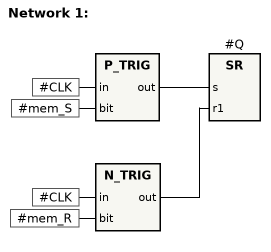
   #_w1 := #CLK AND NOT #mem_S;   // rising edge
   #mem_S := #CLK;
   #_w2 := NOT #CLK AND #mem_R;   // falling edge
   #mem_R := #CLK;
   IF #_w1 THEN
       #Q := TRUE;   // SR flip-flop
   END_IF;
   IF #_w2 THEN #Q := FALSE; END_IF;
END_REGION
END_FUNCTION_BLOCK

FUNCTION_BLOCK "TON_seconds"   // FB8, FBD
{ S7_Optimized_Access := 'TRUE' }
VERSION : 0.1
// stored: AutoNumber true, IsIECCheckEnabled false, IsRetainMemResEnabled false, MemoryReserve 100, SetENOAutomatically false, UDAEnableTagReadback false
   VAR_INPUT
      IN : Bool;
      PT_s : DInt;
   END_VAR
   VAR_OUTPUT
      Q : Bool;
   END_VAR
   VAR
      ton { S7_SetPoint := 'True'} : TON_TIME;
   END_VAR
   VAR_TEMP
      PT : Time;
   END_VAR
BEGIN

REGION Network 1
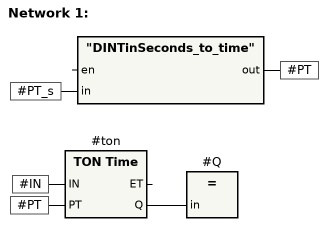
   "DINTinSeconds_to_time"(in := #PT_s, out => #PT);
   #ton(IN := #IN, PT := #PT);   // TON
   #Q := #ton.Q;
END_REGION
END_FUNCTION_BLOCK

FUNCTION_BLOCK "cooling"   // FB17, LAD
{ S7_Optimized_Access := 'TRUE' }
VERSION : 0.1
// stored: AutoNumber true, IsIECCheckEnabled false, IsRetainMemResEnabled false, MemoryReserve 100, SetENOAutomatically false, UDAEnableTagReadback false
   VAR_INPUT
      MagsOn : Bool;
      Work_time_for_CD : Time := T#10m;
   END_VAR
   VAR_OUTPUT
      Vents : Bool;
   END_VAR
   VAR
      IEC_Timer_0_Instance { S7_SetPoint := 'True'} : TON_TIME;
      wasActive : Bool;
   END_VAR
BEGIN

REGION Network 1
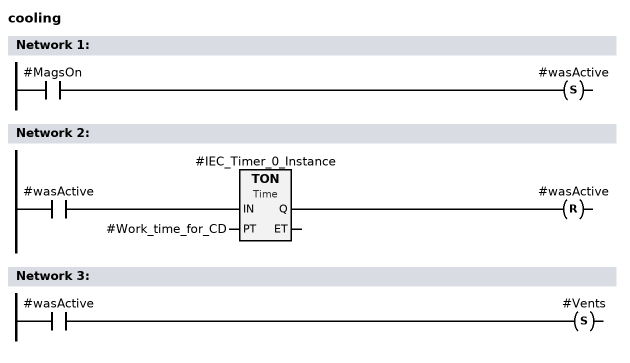
   RUNG wire#powerrail
      Contact( #MagsOn )
      S_Coil( #wasActive )
   END_RUNG
   // the same network as SCL:
   IF #MagsOn THEN #wasActive := TRUE; END_IF;
END_REGION

REGION Network 2
   RUNG wire#powerrail
      Contact( #wasActive )
      { S7_Templates := "time_type := Time" } #IEC_Timer_0_Instance.TON(pt := #Work_time_for_CD, et =>)
      R_Coil( #wasActive )
   END_RUNG
   // the same network as SCL:
   #IEC_Timer_0_Instance(IN := #wasActive, PT := #Work_time_for_CD);   // TON
   IF #IEC_Timer_0_Instance.Q THEN #wasActive := FALSE; END_IF;
END_REGION

REGION Network 3
   RUNG wire#powerrail
      Contact( #wasActive )
      S_Coil( #Vents )
   END_RUNG
   // the same network as SCL:
   IF #wasActive THEN #Vents := TRUE; END_IF;
END_REGION
END_FUNCTION_BLOCK

FUNCTION "LT_GT_OK" : Void   // FC16, FBD
{ S7_Optimized_Access := 'TRUE' }
VERSION : 0.1
// stored: AutoNumber true, IsIECCheckEnabled false, SetENOAutomatically false, UDAEnableTagReadback false
   VAR_INPUT
      value : Real;
      min : Real;
      max : Real;
   END_VAR
   VAR_OUTPUT
      OK : Bool;
      LT_MIN : Bool;
      GT_MAX : Bool;
   END_VAR
BEGIN

REGION Network 1
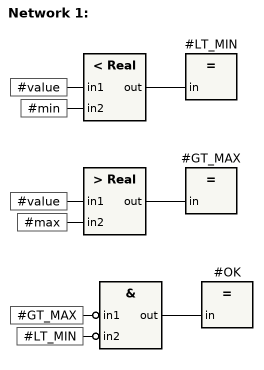
   #LT_MIN := #value < #min;
   #GT_MAX := #value > #max;
   #OK := NOT #GT_MAX AND NOT #LT_MIN;
END_REGION
END_FUNCTION

FUNCTION_BLOCK "execute_semiauto"   // FB46, FBD
{ S7_Optimized_Access := 'TRUE' }
VERSION : 0.1
// stored: AutoNumber true, IsIECCheckEnabled false, IsRetainMemResEnabled false, MemoryReserve 100, SetENOAutomatically false, UDAEnableTagReadback false
   VAR_INPUT
      ALLOWED : Bool;
      xButton : Bool;
      arrived : Bool;
   END_VAR
   VAR_OUTPUT
      y_exec : Bool;
   END_VAR
   VAR
      mem : Bool;
      R_TRIG_Instance { S7_SetPoint := 'True'} : R_TRIG;
      loc : Bool;
   END_VAR
BEGIN

REGION Network 2 (SCL)
   #R_TRIG_Instance(CLK := #xButton);
   IF #ALLOWED THEN
       #y_exec := true;
   (*    IF #R_TRIG_Instance.Q THEN
           IF NOT #arrived THEN
               #y_exec := true;
           ELSE
               #y_exec := false;
           END_IF;
       END_IF; *)
   ELSE
       #y_exec := false;
   END_IF;
END_REGION
END_FUNCTION_BLOCK

FUNCTION_BLOCK "_screen_SetHome"   // FB77, FBD
{ S7_Optimized_Access := 'TRUE' }
VERSION : 0.1
// stored: AutoNumber true, IsIECCheckEnabled false, IsRetainMemResEnabled false, MemoryReserve 100, SetENOAutomatically false, UDAEnableTagReadback false
   VAR
      t_z : "hmi_home_1";
      t_o1 : "hmi_home_1";
      t_o2 : "hmi_home_1";
      t_x : "hmi_home_1";
      t_y : "hmi_home_1";
      z : "hmi_home_1";
      o1 : "hmi_home_1";
      o2 : "hmi_home_1";
      x : "hmi_home_1";
      y : "hmi_home_1";
   END_VAR
BEGIN

REGION Network 1
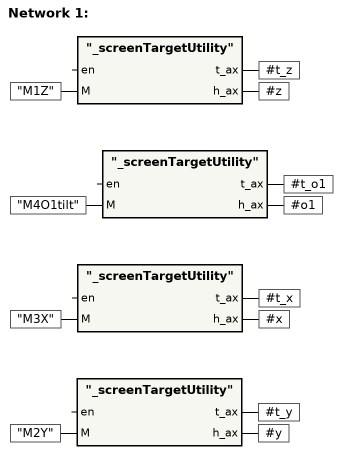
   "_screenTargetUtility"("M" := "M1Z", t_ax => #t_z, h_ax => #z);
   "_screenTargetUtility"("M" := "M4O1tilt", t_ax => #t_o1, h_ax => #o1);
   "_screenTargetUtility"("M" := "M3X", t_ax => #t_x, h_ax => #x);
   "_screenTargetUtility"("M" := "M2Y", t_ax => #t_y, h_ax => #y);
END_REGION

REGION Network 2 (SCL)
   #o2.eF := NOT "M5O2rot".xPredifCal;
   #o2.pos := "M5O2rot".POS;
   #t_o2.pos := "M5O2rot".AMANGRDB.aut_target;
END_REGION
END_FUNCTION_BLOCK

FUNCTION_BLOCK "DelayDirChange"   // FB61, FBD
{ S7_Optimized_Access := 'TRUE' }
VERSION : 0.1
// stored: AutoNumber true, IsIECCheckEnabled false, IsRetainMemResEnabled false, MemoryReserve 100, SetENOAutomatically false, UDAEnableTagReadback false
   VAR_INPUT
      pt : Time := T#2S;
      dirFwd : Bool;
      dirRev : Bool;
   END_VAR
   VAR_OUTPUT
      qFwd : Bool;
      qRev : Bool;
      block : Bool;
   END_VAR
   VAR
      tonfwd { S7_SetPoint := 'True'} : TON_TIME;
      tonrev { S7_SetPoint := 'True'} : TON_TIME;
      block_fwd : Bool;
   END_VAR
   VAR_TEMP
      wait_done : Bool;
      block_rev : Bool;
   END_VAR
BEGIN

REGION Network 2
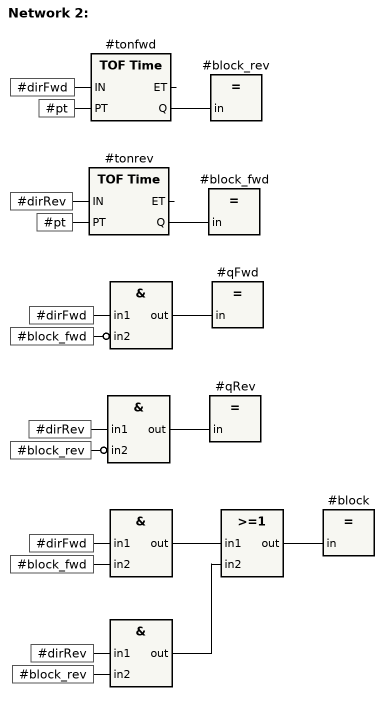
   #tonfwd(IN := #dirFwd, PT := #pt);   // TOF
   #block_rev := #tonfwd.Q;
   #tonrev(IN := #dirRev, PT := #pt);   // TOF
   #block_fwd := #tonrev.Q;
   #qFwd := #dirFwd AND NOT #block_fwd;
   #qRev := #dirRev AND NOT #block_rev;
   #block := (#dirFwd AND #block_fwd) OR (#dirRev AND #block_rev);
END_REGION
END_FUNCTION_BLOCK

FUNCTION_BLOCK "FPDRxMonitorTwoEncodersFB"   // FB63, FBD
{ S7_Optimized_Access := 'TRUE' }
VERSION : 0.1
// stored: AutoNumber true, IsIECCheckEnabled false, IsRetainMemResEnabled false, MemoryReserve 100, SetENOAutomatically false, UDAEnableTagReadback false
   VAR_INPUT
      pos1 { ExternalAccessible := 'False'; ExternalVisible := 'False'; ExternalWritable := 'False'} : Real;
      pos2 { ExternalAccessible := 'False'; ExternalVisible := 'False'; ExternalWritable := 'False'} : Real;
      allowedDelta { ExternalAccessible := 'False'; ExternalVisible := 'False'; ExternalWritable := 'False'} : Real;
      pt : Time;
   END_VAR
   VAR_OUTPUT
      error { ExternalAccessible := 'False'; ExternalVisible := 'False'; ExternalWritable := 'False'} : Bool;
   END_VAR
   VAR
      tonER { S7_SetPoint := 'True'} : TON_TIME;
   END_VAR
   VAR_TEMP
      deltaDangerous : Bool;
   END_VAR
BEGIN

REGION Network 2 (SCL)
   #deltaDangerous := ABS(#pos2 - #pos1)> #allowedDelta;
END_REGION

REGION Network 3
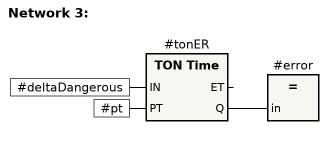
   #tonER(IN := #deltaDangerous, PT := #pt);   // TON
   #error := #tonER.Q;
END_REGION
END_FUNCTION_BLOCK

FUNCTION_BLOCK "Select_remote_or_auto"   // FB24, FBD
{ S7_Optimized_Access := 'TRUE' }
VERSION : 0.1
// stored: AutoNumber true, IsIECCheckEnabled false, IsRetainMemResEnabled false, MemoryReserve 100, SetENOAutomatically false, UDAEnableTagReadback false
BEGIN
END_FUNCTION_BLOCK

FUNCTION_BLOCK "SetA2"   // FB23, FBD
{ S7_Optimized_Access := 'TRUE' }
VERSION : 0.1
// stored: AutoNumber true, IsIECCheckEnabled false, IsRetainMemResEnabled false, MemoryReserve 100, SetENOAutomatically false, UDAEnableTagReadback false
   VAR_INPUT
      xCalibSwMaster : Bool;
      xCalibSwSlave : Bool;
      parMasterCalibPos : Real;
      parSlaveCalibPos : Real;
      btnCopyMasterNow : Bool;
      btnAdjustHorizonPlusStep : Bool;
      btnAdjustHorizonMinusStep : Bool;
      MasterPos : Real;
      SlavePos : Real;
      StepHorAdjust : Real := 10.0;
   END_VAR
   VAR_OUTPUT
      MasterCalibPos : Real;
      MasterCalibNow : Bool;
      SlaveCalibPos : Real;
      SlaveCalibNow : Bool;
   END_VAR
   VAR
      CorrectionFactor : Bool;
      ton { S7_SetPoint := 'True'} : TON_TIME;
      ton1 { S7_SetPoint := 'True'} : TON_TIME;
   END_VAR
BEGIN

REGION Network 1
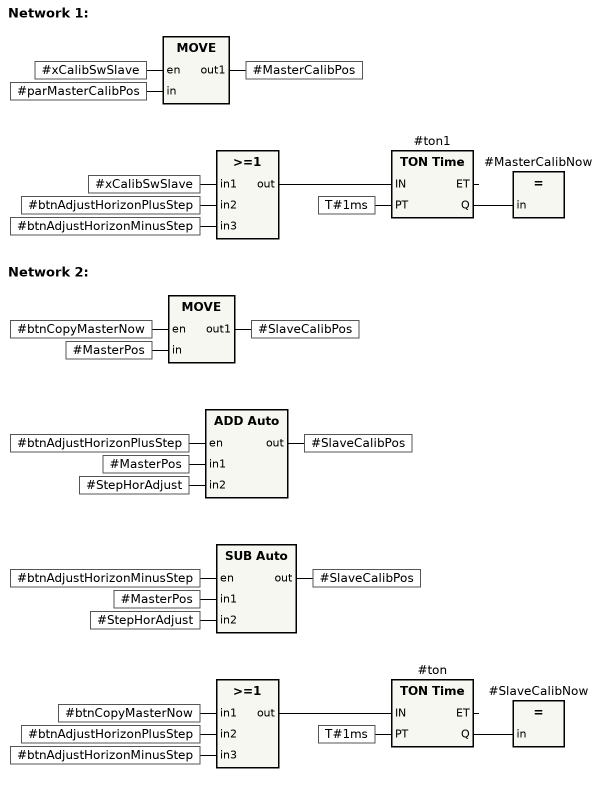
   IF #xCalibSwSlave THEN #MasterCalibPos := #parMasterCalibPos; END_IF;
   #ton1(IN := #xCalibSwSlave OR #btnAdjustHorizonPlusStep OR #btnAdjustHorizonMinusStep, PT := T#1ms);   // TON
   #MasterCalibNow := #ton1.Q;
END_REGION

REGION Network 2
   IF #btnCopyMasterNow THEN #SlaveCalibPos := #MasterPos; END_IF;
   IF #btnAdjustHorizonPlusStep THEN #SlaveCalibPos := #MasterPos + #StepHorAdjust; END_IF;
   IF #btnAdjustHorizonMinusStep THEN #SlaveCalibPos := #MasterPos - #StepHorAdjust; END_IF;
   #ton(IN := #btnCopyMasterNow OR #btnAdjustHorizonPlusStep OR #btnAdjustHorizonMinusStep, PT := T#1ms);   // TON
   #SlaveCalibNow := #ton.Q;
END_REGION
END_FUNCTION_BLOCK

FUNCTION_BLOCK "Slow_inc_quick_drop"   // FB50, FBD
{ S7_Optimized_Access := 'TRUE' }
VERSION : 0.1
// stored: AutoNumber true, IsIECCheckEnabled false, IsRetainMemResEnabled false, MemoryReserve 100, SetENOAutomatically false, UDAEnableTagReadback false
   VAR_INPUT
      ALLOWED : Bool;
      max_v : Real;
      sec_to_max_v : Real;
      req_v : Real;
   END_VAR
   VAR_OUTPUT
      speed : Real;
      er_set { ExternalAccessible := 'False'; ExternalVisible := 'False'; ExternalWritable := 'False'} : Bool;
      wsER : WString;
   END_VAR
   VAR
      accel_v_p_sec : Real;
      accel_per_cycle : Real;
      cycle_time_sec : Real := 0.01;
   END_VAR
BEGIN

REGION Network 2 (SCL)


   #er_set :=  "_MAIN_DB".CLOCK_S_P_SCAN <= 0 OR #sec_to_max_v <=0 ;
   IF #er_set THEN
       #wsER := WSTRING#'ошибка модуля ускорения';
   ELSE
       #wsER := WSTRING#'';
   END_IF;
END_REGION

REGION Network 3 (SCL)
   IF NOT #er_set THEN
       #accel_v_p_sec := #max_v / #sec_to_max_v;
       #accel_per_cycle := #accel_v_p_sec * "_MAIN_DB".CLOCK_S_P_SCAN;
   ELSE
       #accel_per_cycle := 0.0001;
   END_IF;
END_REGION

REGION Network 4 (SCL)
   IF #ALLOWED THEN
       IF NOT #er_set THEN
           IF #req_v > #speed THEN
               #speed := MIN(IN1 := #speed + #accel_per_cycle, IN2 := #req_v);
           ELSIF #req_v < #speed THEN
               #speed := MAX(IN1 := #speed - #accel_per_cycle, IN2 := #req_v);
           END_IF;

       ELSE
           #speed := 0;
       END_IF;
   ELSE
       #speed := 0;
   END_IF;
END_REGION
END_FUNCTION_BLOCK

FUNCTION_BLOCK "auto_digital"   // FB12, FBD
{ S7_Optimized_Access := 'TRUE' }
VERSION : 0.1
// stored: AutoNumber true, IsIECCheckEnabled false, IsRetainMemResEnabled false, MemoryReserve 100, SetENOAutomatically false, UDAEnableTagReadback false
   VAR_INPUT
      ALLOWED : Bool;
      xFwdOK : Bool;
      xRevOK : Bool;
      xFwdFastOK : Bool;
      xRevFastOK : Bool;
   END_VAR
   VAR_OUTPUT
      FWD : Bool;
      REV : Bool;
      QUICK : Bool;
      status_fwd_full : Bool;
      status_mid : Bool;
      status_rev_full : Bool;
   END_VAR
   VAR_IN_OUT
      btn_go_fwd : Bool;
      btn_go_rev : Bool;
   END_VAR
   VAR
      lbs { S7_SetPoint := 'True'} : "last_button_stands";
      mem_fwdok : Bool;
      mem_revok : Bool;
      ton_quick { S7_SetPoint := 'True'} : TON_TIME;
   END_VAR
BEGIN

REGION Network 1
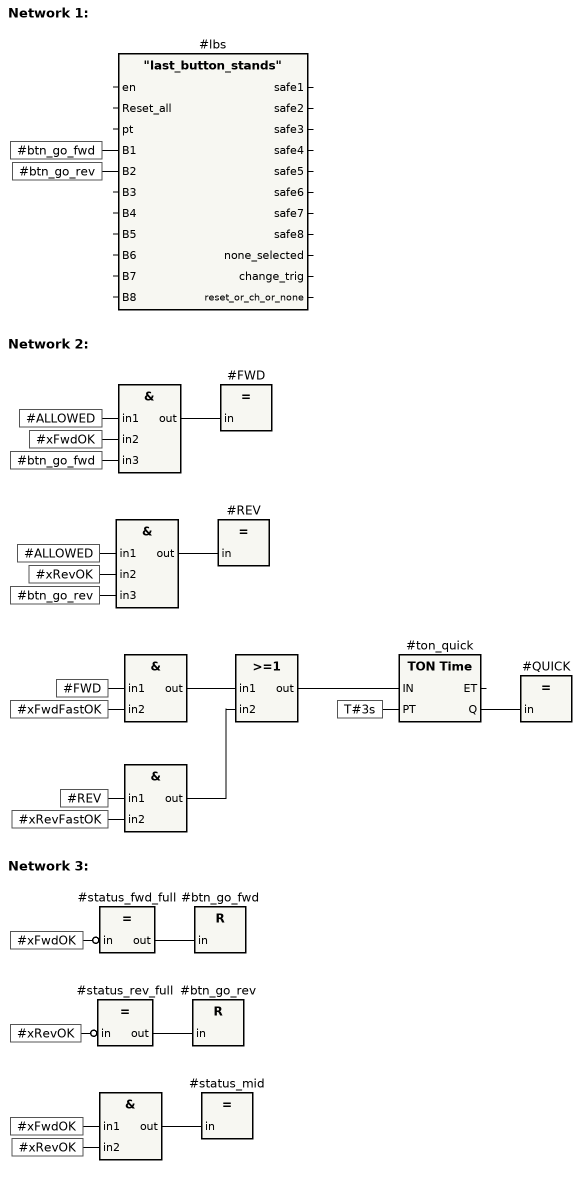
   #lbs(B1 := #btn_go_fwd, B2 := #btn_go_rev);   // "last_button_stands"
END_REGION

REGION Network 2
   #FWD := #ALLOWED AND #xFwdOK AND #btn_go_fwd;
   #REV := #ALLOWED AND #xRevOK AND #btn_go_rev;
   #ton_quick(IN := (#FWD AND #xFwdFastOK) OR (#REV AND #xRevFastOK), PT := T#3s);   // TON
   #QUICK := #ton_quick.Q;
END_REGION

REGION Network 3
   #status_fwd_full := NOT #xFwdOK;
   IF NOT #xFwdOK THEN #btn_go_fwd := FALSE; END_IF;
   #status_rev_full := NOT #xRevOK;
   IF NOT #xRevOK THEN #btn_go_rev := FALSE; END_IF;
   #status_mid := #xFwdOK AND #xRevOK;
END_REGION
END_FUNCTION_BLOCK

FUNCTION "calc_speeds_from_mechanics_1StepperMotor" : Void   // FC33, FBD
{ S7_Optimized_Access := 'TRUE' }
VERSION : 0.1
// stored: AutoNumber true, IsIECCheckEnabled false, SetENOAutomatically false, UDAEnableTagReadback false
   VAR_INPUT
      Vabsmax_deg_per_s : Real;
   END_VAR
   VAR_OUTPUT
      ER_params : Bool;
   END_VAR
   VAR_IN_OUT
      para : "typeMotPara";
   END_VAR
   VAR_TEMP
      counts_per_deg : Real;
      t_acceleration_s : Real;
      "a" : Real;
      v_abs_max : Real;
      t_mx : Real;
      v_min_viable : Real;
      dist_stop : Real;
      dist_auto_done : Real;
      K_min : Real;
      K_min_dist : Real;
      dist_absMax : Real;
   END_VAR
BEGIN

REGION Network 1 (SCL)
   #v_abs_max := #Vabsmax_deg_per_s;
   #t_acceleration_s := #para.t_acc_50Hz_USER;

   #K_min := 0.5 / 50.0;
   #v_min_viable := #v_abs_max * #K_min;

   #t_mx := #t_acceleration_s;
   #ER_params := #t_acceleration_s = 0 OR #v_abs_max = 0 OR #t_mx =0 ;
   IF NOT #ER_params THEN
       #a := #v_abs_max / #t_mx;
       #dist_absMax := #a * #t_mx * #t_mx / 2 + #v_min_viable * #t_mx;
   ELSE
       #a := 0;
        #dist_absMax := 999;
   END_IF;
   #K_min_dist :=0.5/ 50.0 ;//#K_min * 0.8;
   #dist_stop := #dist_absMax * #K_min_dist;
   #dist_auto_done := #dist_stop * 1.2;
END_REGION

REGION Network 2 (SCL)
   //#para.dist_absMax_LOGIC := #dist_fast;
   #para.dist_stop_USER := #dist_stop;
   #para.dist_auto_done_LOGIC := #dist_auto_done;
   //#para.dist_auto_maxCor_LOGIC := 0.1 * #para.dist_absMax_LOGIC;
   #para.v_absoluteMax_LOGIC := #v_abs_max;
   #para.v_crawl_USER := #v_min_viable;
   //#para.v_auto_maxCor_LOGIC := 0.1 * #para.v_absoluteMax_LOGIC;
END_REGION
END_FUNCTION

FUNCTION "calc_speeds_from_mechanics_2SyncedDrivesTUBEZ" : Void   // FC25, FBD
{ S7_Optimized_Access := 'TRUE' }
VERSION : 0.1
// stored: AutoNumber true, IsIECCheckEnabled false, SetENOAutomatically false, UDAEnableTagReadback false
   VAR_INPUT
      mm_per_outputshaft_rev : Real;
      reduction_ration : Real;
      max_revs_at_10V : Real;
      counts_per_encoder_rev : Real;
      encoder_placed_on_motor : Bool;
   END_VAR
   VAR_OUTPUT
      Vabsmax_mm_per_s : Real;
      counts_per_mm : Real;
      ER_params : Bool;
   END_VAR
   VAR_IN_OUT
      para : "typeMotPara";
   END_VAR
   VAR_TEMP
      t_acceleration_s : Real;
      maxV_mm_per_min : Real;
      "a" : Real;
      v_abs_max : Real;
      t_mx : Real;
      dist_fast : Real;
      v_min_viable : Real;
      dist_stop : Real;
      dist_auto_done : Real;
      K_min : Real;
      K_min_dist : Real;
      dist_absMax : Real;
      t_fst : Real;
      v_fast : Real;
   END_VAR
BEGIN

REGION Network 2 (SCL)

   #maxV_mm_per_min := #max_revs_at_10V / #reduction_ration * #mm_per_outputshaft_rev;

   #Vabsmax_mm_per_s := #maxV_mm_per_min / 60;
END_REGION

REGION Network 3 (SCL)
   IF #encoder_placed_on_motor THEN
       #counts_per_mm :=  #counts_per_encoder_rev * #reduction_ration / #mm_per_outputshaft_rev  ;
   ELSE
       #counts_per_mm := #counts_per_encoder_rev /  #mm_per_outputshaft_rev;

   END_IF;
END_REGION

REGION Network 4 (SCL)
   #v_abs_max := #Vabsmax_mm_per_s;
   #t_acceleration_s := #para.t_acc_50Hz_USER;
   #v_fast := #para.v_absoluteMax_LOGIC;

   #K_min := 1.0/50.0;
   #v_min_viable := #v_abs_max * #K_min;

   #t_mx := #t_acceleration_s;
   #ER_params := #t_acceleration_s = 0 OR #v_abs_max = 0 OR #t_mx =0 ;
   IF NOT #ER_params THEN
       #t_fst := #t_acceleration_s * #v_fast / #v_abs_max;
       #a := #v_abs_max / #t_mx;
       #dist_absMax := #a * #t_mx * #t_mx / 2 + #v_min_viable * #t_mx;
       #dist_fast := #a * #t_fst * #t_fst / 2 + #v_min_viable * #t_fst;
   ELSE
       #a := 0;
       #dist_fast := #dist_absMax := 999;
       #t_fst := 0;
   END_IF;
   #K_min_dist := 1.0/ 50.0;//#K_min * 0.8;
   #dist_stop := #dist_absMax * #K_min_dist;
   #dist_auto_done := #dist_stop * 4.0;//1.4;//.0;// 1.2;
END_REGION

REGION Network 5 (SCL)
   #para.dist_absMax_LOGIC := #dist_fast;
   #para.dist_stop_USER := #dist_stop;
   #para.dist_auto_done_LOGIC := #dist_auto_done;
   #para.v_absoluteMax_LOGIC := #v_abs_max;
   #para.v_crawl_USER := #v_min_viable;
END_REGION
END_FUNCTION

FUNCTION_BLOCK "encoder2"   // FB62, FBD
{ S7_Optimized_Access := 'TRUE' }
VERSION : 0.1
// stored: AutoNumber true, IsIECCheckEnabled false, IsRetainMemResEnabled false, MemoryReserve 100, SetENOAutomatically false, UDAEnableTagReadback false
   VAR_INPUT
      xCal : Bool;
      ENC : Real;
      posCal : Real;
   END_VAR
   VAR_OUTPUT
      i_times_cal : Int;
      retain_test : Bool;
      POS : Real;
   END_VAR
   VAR
      xCal_filtered : Bool;
      not_first_scan : Bool;
      offset : Real;
   END_VAR
   VAR RETAIN
      MEM : Real;
   END_VAR
   VAR
      xCal_mem : Bool;
   END_VAR
   VAR RETAIN
      calibrated : Bool;
   END_VAR
   VAR
      ton_block_calib { S7_SetPoint := 'True'} : TON_TIME;
      tonFilter { S7_SetPoint := 'True'} : TON_TIME;
   END_VAR
BEGIN

REGION Network 1
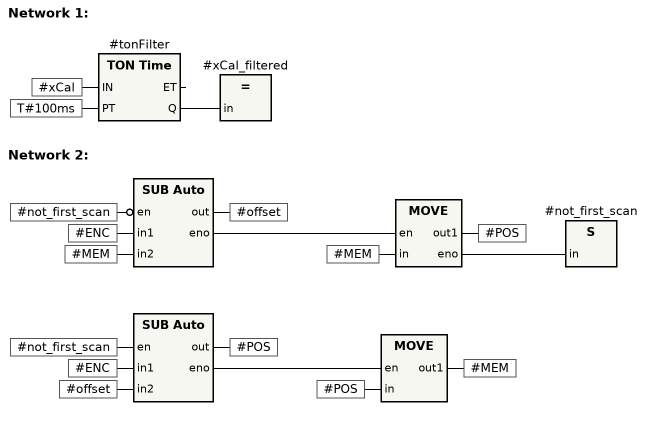
   #tonFilter(IN := #xCal, PT := T#100ms);   // TON
   #xCal_filtered := #tonFilter.Q;
END_REGION

REGION Network 2
   IF NOT #not_first_scan THEN
       #offset := #ENC - #MEM;
       #POS := #MEM;
       #not_first_scan := TRUE;
   END_IF;
   IF #not_first_scan THEN
       #POS := #ENC - #offset;
       #MEM := #POS;
   END_IF;
END_REGION

REGION Network 3 (SCL)
   IF #xCal_filtered AND NOT #xCal_mem THEN
       #offset := #ENC - #posCal;
       #calibrated := true;
       #i_times_cal := #i_times_cal + 1;
   END_IF;
   #xCal_mem := #xCal_filtered;
END_REGION
END_FUNCTION_BLOCK

FUNCTION_BLOCK "encoderMesSpeed"   // FB19, FBD
{ S7_Optimized_Access := 'TRUE' }
VERSION : 0.1
// stored: AutoNumber true, IsIECCheckEnabled false, IsRetainMemResEnabled false, MemoryReserve 100, SetENOAutomatically false, UDAEnableTagReadback false
BEGIN
END_FUNCTION_BLOCK

FUNCTION_BLOCK "encoder_mes_speed"   // FB20, FBD
{ S7_Optimized_Access := 'TRUE' }
VERSION : 0.1
// stored: AutoNumber true, IsIECCheckEnabled false, IsRetainMemResEnabled false, MemoryReserve 100, SetENOAutomatically false, UDAEnableTagReadback false
   VAR_INPUT
      Cycle_Time_s : Real;
      Pos : Real;
   END_VAR
   VAR_OUTPUT
      Speed_mm_p_sec : Real;
   END_VAR
   VAR
      MEM : LReal;
      RET_VAL : LReal;
      Pos_was : Real;
   END_VAR
   VAR_TEMP
      Speed_mm_p_sec_temp : Real;
      delta : Real;
      n : Real;
   END_VAR
BEGIN

REGION Network 1
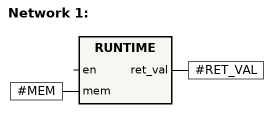
   // no SCL statement known for Runtime: written as a call
   #RET_VAL := Runtime(mem := #MEM);
END_REGION

REGION Network 2 (SCL)
   #delta := #Pos - #Pos_was;
   #Speed_mm_p_sec_temp := #delta / #Cycle_Time_s;
   #n := 10;
   #Speed_mm_p_sec := (#Speed_mm_p_sec * (#n - 1) + #Speed_mm_p_sec_temp)/ #n;

   #Pos_was := #Pos;
END_REGION
END_FUNCTION_BLOCK

FUNCTION_BLOCK "manual_digital"   // FB13, FBD
{ S7_Optimized_Access := 'TRUE' }
VERSION : 0.1
// stored: AutoNumber true, IsIECCheckEnabled false, IsRetainMemResEnabled false, MemoryReserve 100, SetENOAutomatically false, UDAEnableTagReadback false
   VAR_INPUT
      ALLOWED : Bool;
      xFwdOk : Bool;
      xRevOk : Bool;
      xFwdFastOK : Bool;
      xRevFastOK : Bool;
   END_VAR
   VAR_OUTPUT
      FWD : Bool;
      REV : Bool;
      FAST : Bool;
   END_VAR
   VAR_IN_OUT
      btn_FWD : Bool;
      btn_REV : Bool;
   END_VAR
   VAR
      lbs { S7_SetPoint := 'True'} : "last_button_stands";
      ton_quick { S7_SetPoint := 'True'} : TON_TIME;
   END_VAR
BEGIN

REGION Network 1
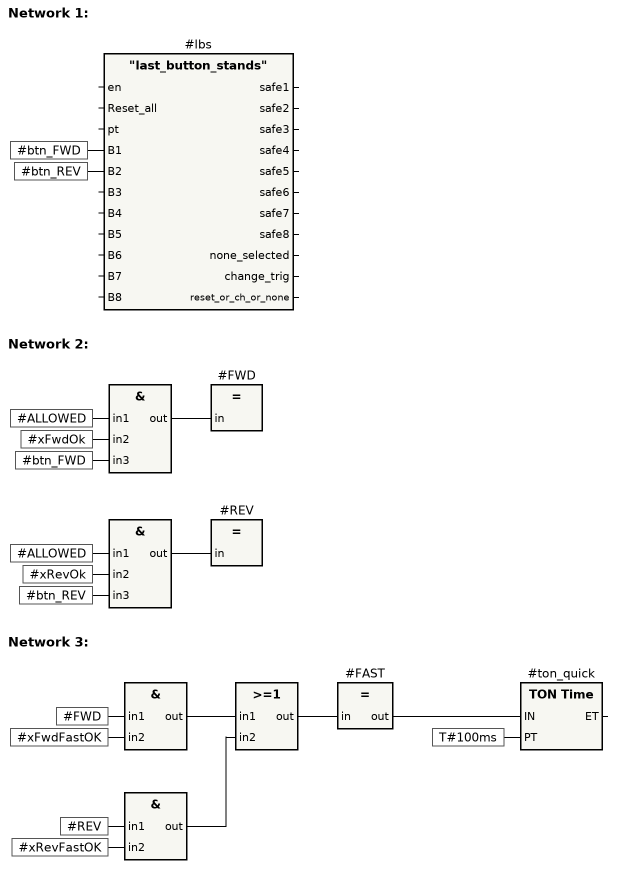
   #lbs(B1 := #btn_FWD, B2 := #btn_REV);   // "last_button_stands"
END_REGION

REGION Network 2
   #FWD := #ALLOWED AND #xFwdOk AND #btn_FWD;
   #REV := #ALLOWED AND #xRevOk AND #btn_REV;
END_REGION

REGION Network 3
   #FAST := (#FWD AND #xFwdFastOK) OR (#REV AND #xRevFastOK);
   #ton_quick(IN := #FAST, PT := T#100ms);   // TON
END_REGION
END_FUNCTION_BLOCK

FUNCTION_BLOCK "monitor_sw_no_encoder"   // FB36, FBD
{ S7_Optimized_Access := 'TRUE' }
VERSION : 0.1
// stored: AutoNumber true, IsIECCheckEnabled false, IsRetainMemResEnabled false, MemoryReserve 100, SetENOAutomatically false, UDAEnableTagReadback false
   VAR_INPUT
      xFWD : Bool;
      xFWDSLO : Bool;
      xREVSLO : Bool;
      xREV : Bool;
      go_FWD : Bool;
      go_REV : Bool;
      para_slo_to_slo : Time := T#2m;
      para_slo_to_end : Time := T#1m;
   END_VAR
   VAR_OUTPUT
      ER_FWD : Bool;
      ER_FWDSLO : Bool;
      ER_REVSLO : Bool;
      ER_REV : Bool;
   END_VAR
   VAR
      ton_fwd { S7_SetPoint := 'True'} : TON_TIME;
      ton_rev { S7_SetPoint := 'True'} : TON_TIME;
      ton_fwdslo { S7_SetPoint := 'True'} : TON_TIME;
      ton_revslo { S7_SetPoint := 'True'} : TON_TIME;
   END_VAR
BEGIN

REGION Network 1
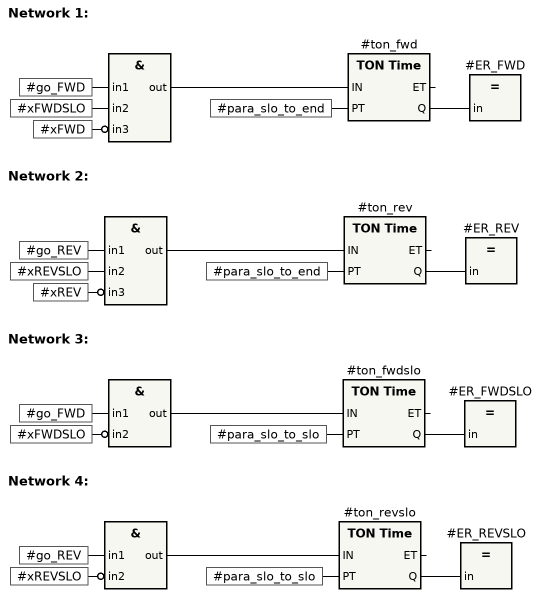
   #ton_fwd(IN := #go_FWD AND #xFWDSLO AND NOT #xFWD, PT := #para_slo_to_end);   // TON
   #ER_FWD := #ton_fwd.Q;
END_REGION

REGION Network 2
   #ton_rev(IN := #go_REV AND #xREVSLO AND NOT #xREV, PT := #para_slo_to_end);   // TON
   #ER_REV := #ton_rev.Q;
END_REGION

REGION Network 3
   #ton_fwdslo(IN := #go_FWD AND NOT #xFWDSLO, PT := #para_slo_to_slo);   // TON
   #ER_FWDSLO := #ton_fwdslo.Q;
END_REGION

REGION Network 4
   #ton_revslo(IN := #go_REV AND NOT #xREVSLO, PT := #para_slo_to_slo);   // TON
   #ER_REVSLO := #ton_revslo.Q;
END_REGION
END_FUNCTION_BLOCK

FUNCTION "mot_auto_calc_arrived" : Void   // FC17, FBD
{ S7_Optimized_Access := 'TRUE' }
VERSION : 0.1
// stored: AutoNumber true, IsIECCheckEnabled false, SetENOAutomatically false, UDAEnableTagReadback false
   VAR_INPUT
      Target : Real;
      Pos : Real;
      Modifier_delta : Real;
      par_prec_au : Real;
      par_dist_stop : Real;
   END_VAR
   VAR_OUTPUT
      arrived : Bool;
      distance : Real;
      stop_now : Bool;
   END_VAR
BEGIN

REGION Network 2 (SCL)
   #distance := #Target - (#Pos+#Modifier_delta);

   #arrived := ABS(#distance) <= #par_prec_au;

   #stop_now := ABS(#distance) <= #par_dist_stop;
END_REGION
END_FUNCTION

FUNCTION "mot_inertia_speed" : Void   // FC27, FBD
{ S7_Optimized_Access := 'TRUE' }
VERSION : 0.1
// stored: AutoNumber true, IsIECCheckEnabled false, SetENOAutomatically false, UDAEnableTagReadback false
   VAR_INPUT
      set_speed : Real;
      par : "typeMotPara";
      seconds_per_clock : Real;
   END_VAR
   VAR_OUTPUT
      ER_SET : Bool;
   END_VAR
   VAR_IN_OUT
      speed : Real;
   END_VAR
   VAR_TEMP
      v_delta : Real;
      v_step_per_cycle_max : Real;
      abs_max_speed : Real;
      time_abs_max : Real;
   END_VAR
BEGIN

REGION Network 2 (SCL)
   #v_delta := ABS(#speed - #set_speed);
   #abs_max_speed := #par.v_absoluteMax_LOGIC;
   #time_abs_max := #par.t_acc_50Hz_USER;
   #ER_SET := #abs_max_speed <= 0 OR #time_abs_max <= 0 OR #seconds_per_clock <= 0;

   #v_step_per_cycle_max := #abs_max_speed / #time_abs_max * #seconds_per_clock;
   IF #ER_SET THEN
       #speed := 0;
   ELSE
       IF #v_delta < #v_step_per_cycle_max THEN
           #speed := #set_speed;
       ELSE
           IF #set_speed > #speed THEN
               #speed := #speed + #v_step_per_cycle_max;
           ELSE
               #speed := #speed - #v_step_per_cycle_max;
           END_IF;
       END_IF;
   END_IF;
END_REGION
END_FUNCTION

FUNCTION_BLOCK "p_trig_to_set_reset"   // FB38, FBD
{ S7_Optimized_Access := 'TRUE' }
VERSION : 0.1
// stored: AutoNumber true, IsIECCheckEnabled false, IsRetainMemResEnabled false, MemoryReserve 100, SetENOAutomatically false, UDAEnableTagReadback false
   VAR_INPUT
      "DO" : Bool;
   END_VAR
   VAR_OUTPUT
      DONE : Bool;
   END_VAR
   VAR_IN_OUT
      inout_button : Bool;
   END_VAR
   VAR
      mem_1 : Bool;
      mem_2 : Bool;
   END_VAR
   VAR_TEMP   // added for the SCL form of the ladder/FBD networks
      _w1 : Bool;
      _w2 : Bool;
   END_VAR
BEGIN

REGION Network 1
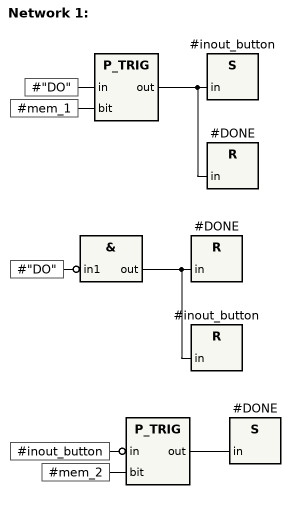
   #_w1 := #"DO" AND NOT #mem_1;   // rising edge
   #mem_1 := #"DO";
   IF #_w1 THEN
       #inout_button := TRUE;
       #DONE := FALSE;
   END_IF;
   IF NOT #"DO" THEN
       #DONE := FALSE;
       #inout_button := FALSE;
   END_IF;
   #_w2 := NOT #inout_button AND NOT #mem_2;   // rising edge
   #mem_2 := NOT #inout_button;
   IF #_w2 THEN #DONE := TRUE; END_IF;
END_REGION
END_FUNCTION_BLOCK

FUNCTION "select_remote" : Void   // FC36, FBD
{ S7_Optimized_Access := 'TRUE' }
VERSION : 0.1
// stored: AutoNumber true, IsIECCheckEnabled false, SetENOAutomatically false, UDAEnableTagReadback false
   VAR_INPUT
      MD_AUtO : Bool;
      MD_DESK : Bool;
      MD_RC : Bool;
      MD_RC_override : Bool;
      Joystick : Real;
      speed_RCfast : Real;
      speed_RCOverride : Real;
   END_VAR
   VAR_OUTPUT
      speed : Real;
   END_VAR
   VAR_IN_OUT
      m_AUTO : Bool;
      m_MAN : Bool;
      m_override : Bool;
   END_VAR
   VAR_TEMP
      slow_speed_static : Real;
      fast_speed_static : Real;
   END_VAR
BEGIN

REGION Network 2
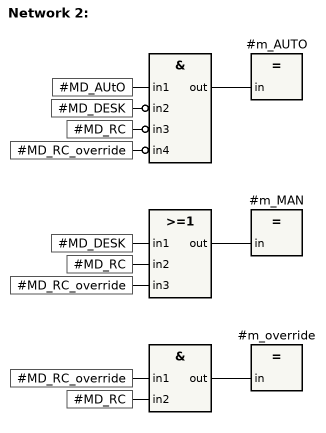
   #m_AUTO := #MD_AUtO AND NOT #MD_DESK AND NOT #MD_RC AND NOT #MD_RC_override;
   #m_MAN := #MD_DESK OR #MD_RC OR #MD_RC_override;
   #m_override := #MD_RC_override AND #MD_RC;
END_REGION
END_FUNCTION

FUNCTION_BLOCK "select_remoteFB"   // FB16, LAD
{ S7_Optimized_Access := 'TRUE' }
VERSION : 0.1
// stored: AutoNumber true, IsIECCheckEnabled false, IsRetainMemResEnabled false, MemoryReserve 100, SetENOAutomatically false, UDAEnableTagReadback false
   VAR_INPUT
      MD_AUtO : Bool;
      MD_DESK { ExternalAccessible := 'False'; ExternalVisible := 'False'; ExternalWritable := 'False'} : Bool;
      MD_RC { ExternalAccessible := 'False'; ExternalVisible := 'False'; ExternalWritable := 'False'} : Bool;
      MD_RC_override : Bool;
      Joystick { ExternalAccessible := 'False'; ExternalVisible := 'False'; ExternalWritable := 'False'} : Real;
      speed_RCfast { ExternalAccessible := 'False'; ExternalVisible := 'False'; ExternalWritable := 'False'} : Real;
      speed_RCOverride { ExternalAccessible := 'False'; ExternalVisible := 'False'; ExternalWritable := 'False'} : Real;
   END_VAR
   VAR_OUTPUT
      m_AUTO : Bool;
      m_MAN : Bool;
      m_override : Bool;
      speed { ExternalAccessible := 'False'; ExternalVisible := 'False'; ExternalWritable := 'False'} : Real;
   END_VAR
   VAR_TEMP
      slow_speed_static : Real;
      fast_speed_static : Real;
   END_VAR
BEGIN

REGION Network 1
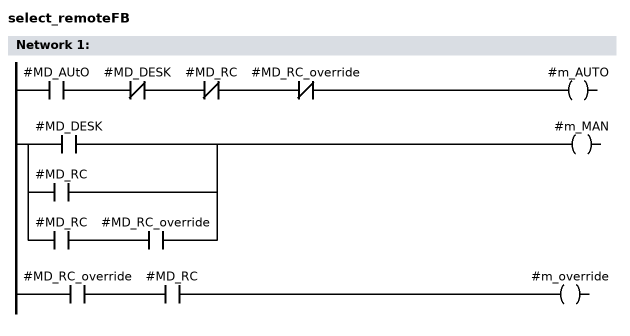
   RUNG wire#powerrail
      Contact( #MD_AUtO )
      I_Contact( #MD_DESK )
      I_Contact( #MD_RC )
      I_Contact( #MD_RC_override )
      Coil( #m_AUTO )
   END_RUNG
   RUNG wire#powerrail
      Contact( #MD_DESK )
      wire#w1
      Coil( #m_MAN )
   END_RUNG
   RUNG wire#powerrail
      Contact( #MD_RC )
   END_RUNG wire#w1
   RUNG wire#powerrail
      Contact( #MD_RC )
      Contact( #MD_RC_override )
   END_RUNG wire#w1
   RUNG wire#powerrail
      Contact( #MD_RC_override )
      Contact( #MD_RC )
      Coil( #m_override )
   END_RUNG
   // the same network as SCL:
   #m_AUTO := #MD_AUtO AND NOT #MD_DESK AND NOT #MD_RC AND NOT #MD_RC_override;
   #m_MAN := #MD_DESK OR #MD_RC OR (#MD_RC AND #MD_RC_override);
   #m_override := #MD_RC_override AND #MD_RC;
END_REGION
END_FUNCTION_BLOCK

FUNCTION_BLOCK "select_remoteMP_FB"   // FB60, LAD
{ S7_Optimized_Access := 'TRUE' }
VERSION : 0.1
// stored: AutoNumber true, IsIECCheckEnabled false, IsRetainMemResEnabled false, MemoryReserve 100, SetENOAutomatically false, UDAEnableTagReadback false
   VAR_INPUT
      MD_AUtO : Bool;
      MD_DESK { ExternalAccessible := 'False'; ExternalVisible := 'False'; ExternalWritable := 'False'} : Bool;
      MD_RC { ExternalAccessible := 'False'; ExternalVisible := 'False'; ExternalWritable := 'False'} : Bool;
      Joystick { ExternalAccessible := 'False'; ExternalVisible := 'False'; ExternalWritable := 'False'} : Real;
      speed_RCfast { ExternalAccessible := 'False'; ExternalVisible := 'False'; ExternalWritable := 'False'} : Real;
   END_VAR
   VAR_OUTPUT
      speed { ExternalAccessible := 'False'; ExternalVisible := 'False'; ExternalWritable := 'False'} : Real;
   END_VAR
   VAR_IN_OUT
      m_AUTO : Bool;
      m_MAN : Bool;
   END_VAR
   VAR_TEMP
      slow_speed_static : Real;
      fast_speed_static : Real;
   END_VAR
BEGIN

REGION Network 1
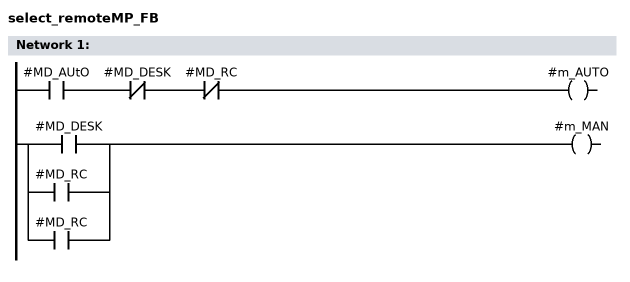
   RUNG wire#powerrail
      Contact( #MD_AUtO )
      I_Contact( #MD_DESK )
      I_Contact( #MD_RC )
      Coil( #m_AUTO )
   END_RUNG
   RUNG wire#powerrail
      Contact( #MD_DESK )
      wire#w1
      Coil( #m_MAN )
   END_RUNG
   RUNG wire#powerrail
      Contact( #MD_RC )
   END_RUNG wire#w1
   RUNG wire#powerrail
      Contact( #MD_RC )
   END_RUNG wire#w1
   // the same network as SCL:
   #m_AUTO := #MD_AUtO AND NOT #MD_DESK AND NOT #MD_RC;
   #m_MAN := #MD_DESK OR #MD_RC OR #MD_RC;
END_REGION
END_FUNCTION_BLOCK

FUNCTION_BLOCK "MAN_DESCRETE_cycle"   // FB41, FBD
{ S7_Optimized_Access := 'TRUE' }
VERSION : 0.1
// stored: AutoNumber true, IsIECCheckEnabled false, IsRetainMemResEnabled false, MemoryReserve 100, SetENOAutomatically false, UDAEnableTagReadback false
   VAR_INPUT
      off_conditions : Bool;
      on_trigger : Bool;
   END_VAR
   VAR_OUTPUT
      motors_go_now_command : Bool;
   END_VAR
   VAR_IN_OUT
      sate : UInt;
   END_VAR
BEGIN

REGION Network 1
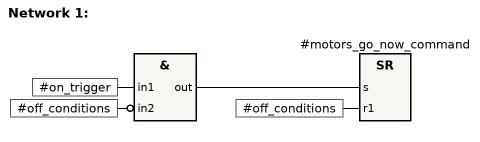
   IF #on_trigger AND NOT #off_conditions THEN
       #motors_go_now_command := TRUE;   // SR flip-flop
   END_IF;
   IF #off_conditions THEN #motors_go_now_command := FALSE; END_IF;
END_REGION
END_FUNCTION_BLOCK

FUNCTION_BLOCK "man_descrete_sr"   // FB28, FBD
{ S7_Optimized_Access := 'TRUE' }
VERSION : 0.1
// stored: AutoNumber true, IsIECCheckEnabled false, IsRetainMemResEnabled false, MemoryReserve 100, SetENOAutomatically false, UDAEnableTagReadback false
   VAR_INPUT
      condions : Bool;
      buttons : Bool;
      arrived : Bool;
   END_VAR
   VAR_OUTPUT
      exce_man : Bool;
   END_VAR
BEGIN

REGION Network 1
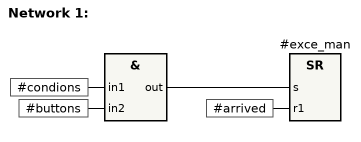
   IF #condions AND #buttons THEN
       #exce_man := TRUE;   // SR flip-flop
   END_IF;
   IF #arrived THEN #exce_man := FALSE; END_IF;
END_REGION
END_FUNCTION_BLOCK

FUNCTION "ER_lim_auto_ws" : Void   // FC19, FBD
{ S7_Optimized_Access := 'TRUE' }
VERSION : 0.1
// stored: AutoNumber true, IsIECCheckEnabled false, SetENOAutomatically false, UDAEnableTagReadback false
   VAR_INPUT
      par_fwd_limit : Real;
      par_rev_limit : Real;
      par_dist_fast : Real;
      par_spd_fast : Real;
      par_spd_slow : Real;
   END_VAR
   VAR_OUTPUT
      ER_settings : Bool;
      wsER : WString;
   END_VAR
   VAR_TEMP
      tmp_fwdLEREV : Bool;
      tmp_fastL0 : Bool;
      tmp_fastLEslo : Bool;
   END_VAR
BEGIN

REGION Network 1
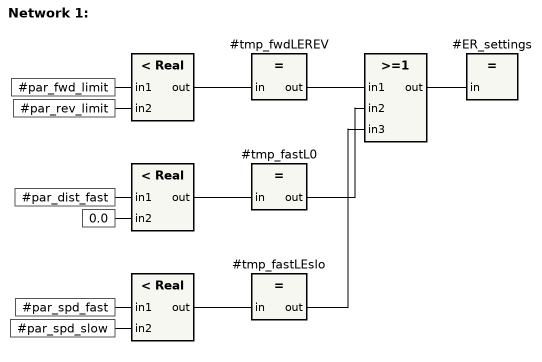
   #tmp_fwdLEREV := #par_fwd_limit < #par_rev_limit;
   #tmp_fastL0 := #par_dist_fast < 0.0;
   #tmp_fastLEslo := #par_spd_fast < #par_spd_slow;
   #ER_settings := #tmp_fwdLEREV OR #tmp_fastL0 OR #tmp_fastLEslo;
END_REGION

REGION Network 2 (SCL)
   IF #tmp_fwdLEREV THEN
       #wsER := WSTRING#'lim fwd LE rev';
   END_IF;
   IF #tmp_fastL0 THEN
       #wsER := WSTRING#'dist fast 0';
   END_IF;
   IF #tmp_fastLEslo THEN
       #wsER := WSTRING#'v fast LE slo';
   END_IF;
END_REGION
END_FUNCTION

FUNCTION "ER_lim_v_ws" : Void   // FC20, FBD
{ S7_Optimized_Access := 'TRUE' }
VERSION : 0.1
// stored: AutoNumber true, IsIECCheckEnabled false, SetENOAutomatically false, UDAEnableTagReadback false
   VAR_INPUT
      v_auto_USER : Real;
      v_absoluteMax_LOGIC : Real;
      v_fast_USER : Real;
      v_blind_USER : Real;
      v_crawl_LOGIC : Real;
   END_VAR
   VAR_OUTPUT
      ER_settings : Bool;
      wsER : WString;
   END_VAR
   VAR_TEMP
      tmp_fwdLEREV : Bool;
      tmp_fastL0 : Bool;
      tmp_fastLEslo : Bool;
      e_v_auto : Bool;
      e_v_blind : Bool;
      e_v_crawl : Bool;
      e_v_fast : Bool;
   END_VAR
BEGIN

REGION Network 1
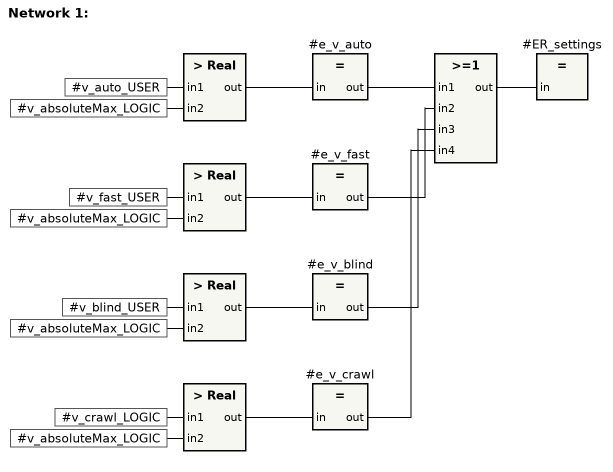
   #e_v_auto := #v_auto_USER > #v_absoluteMax_LOGIC;
   #e_v_fast := #v_fast_USER > #v_absoluteMax_LOGIC;
   #e_v_blind := #v_blind_USER > #v_absoluteMax_LOGIC;
   #e_v_crawl := #v_crawl_LOGIC > #v_absoluteMax_LOGIC;
   #ER_settings := #e_v_auto OR #e_v_fast OR #e_v_blind OR #e_v_crawl;
END_REGION

REGION Network 2 (SCL)
   IF #e_v_auto THEN
       #wsER := WSTRING#'v auto GT abs max';
   END_IF;
   IF #e_v_fast THEN
       #wsER := WSTRING#'v fast GT abs max';
   END_IF;
   IF #e_v_blind THEN
       #wsER := WSTRING#'v blind GT abs max';
   END_IF;
   IF #e_v_crawl THEN
       #wsER := WSTRING#'v crawl GT abs max';
   END_IF;
END_REGION
END_FUNCTION

FUNCTION "FilmInSafeZoneDeterminator" : Void   // FC18, FBD
{ S7_Optimized_Access := 'TRUE' }
VERSION : 0.1
// stored: AutoNumber true, IsIECCheckEnabled false, SetENOAutomatically false, UDAEnableTagReadback false
   VAR_INPUT
      X : Real;
      x_min : Real;
      x_max : Real;
      Y : Real;
      y_min : Real;
      y_max : Real;
      FILM_MODE : Bool;
      par_dist_arrived : Real;
   END_VAR
   VAR_OUTPUT
      WITHIN_SAFE_ZONE : Bool;
   END_VAR
   VAR_TEMP
      loc_x_safe : Bool;
      loc_y_safe : Bool;
      loc_is_safe : Bool;
      x_min_loc : Real;
      x_max_loc : Real;
      y_min_loc : Real;
      y_max_loc : Real;
      loc_par_dist_arrived : Real;
   END_VAR
BEGIN

REGION Network 2 (SCL)
   #loc_par_dist_arrived := 3 * #par_dist_arrived;

   #x_min_loc := #x_min - #loc_par_dist_arrived;
   #x_max_loc := #x_max + #loc_par_dist_arrived;

   #y_min_loc := #y_min - #loc_par_dist_arrived;
   #y_max_loc := #y_max + #loc_par_dist_arrived;
END_REGION

REGION Network 3
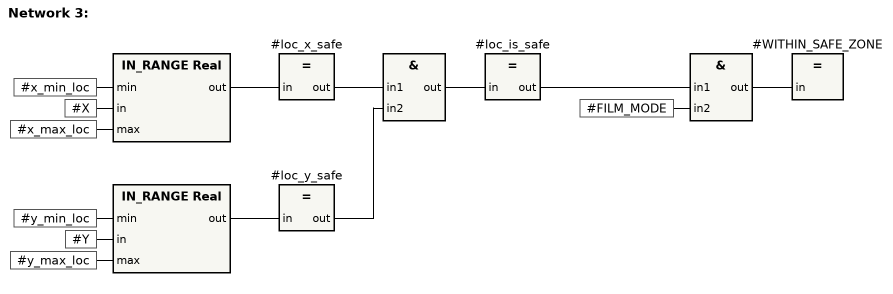
   #loc_x_safe := (#x_min_loc <= #X) AND (#X <= #x_max_loc);
   #loc_y_safe := (#y_min_loc <= #Y) AND (#Y <= #y_max_loc);
   #loc_is_safe := #loc_x_safe AND #loc_y_safe;
   #WITHIN_SAFE_ZONE := #loc_is_safe AND #FILM_MODE;
END_REGION
END_FUNCTION

FUNCTION_BLOCK "cycle_point_to_point"   // FB51, FBD
{ S7_Optimized_Access := 'TRUE' }
VERSION : 0.1
// stored: AutoNumber true, IsIECCheckEnabled false, IsRetainMemResEnabled false, MemoryReserve 100, SetENOAutomatically false, UDAEnableTagReadback false
   VAR
      saved_points : Bool;
      defect_points : Bool;
   END_VAR
BEGIN
END_FUNCTION_BLOCK

FUNCTION_BLOCK "P_TRIG"
{ S7_Optimized_Access := 'FALSE' }
VERSION : 0.1
   VAR_INPUT 
      IN : Bool;
   END_VAR

   VAR_OUTPUT 
      P : Bool;
      N : Bool;
   END_VAR

   VAR 
      WAS : Bool;
   END_VAR


BEGIN
	#P := #IN AND NOT #WAS;
	#N := NOT #IN AND #WAS;
	#WAS := #IN;
END_FUNCTION_BLOCK

FUNCTION_BLOCK "P_TRIG_1"
{ S7_Optimized_Access := 'FALSE' }
VERSION : 0.1
   VAR_INPUT 
      IN : Bool;
   END_VAR

   VAR_OUTPUT 
      P : Bool;
      N : Bool;
   END_VAR

   VAR 
      WAS : Bool;
   END_VAR


BEGIN
	#P := #IN AND NOT #WAS;
	#N := NOT #IN AND #WAS;
	#WAS := #IN;
END_FUNCTION_BLOCK

FUNCTION_BLOCK "TRIG_MULTI"
{ S7_Optimized_Access := 'TRUE' }
VERSION : 0.1
   VAR_INPUT 
      IN : Bool;
      allowed_on : Bool := TRUE;
      allowed_change : Bool := TRUE;
   END_VAR

   VAR_OUTPUT 
      P : Bool;
      N : Bool;
      changed : Bool;
   END_VAR

   VAR_IN_OUT 
      SR : Bool;
      RS : Bool;
      S : Bool;
      R : Bool;
      INVERT : Bool;
   END_VAR

   VAR 
      tr : "P_TRIG";
      tr_al : "P_TRIG";
   END_VAR


BEGIN
	
	#tr(IN:=#IN );
	#tr_al(IN := #allowed_on);
	#P := #tr.P AND #allowed_on;
	IF #P AND #allowed_change THEN
	    #SR := true;
	    #RS := false;
	    #S := true;
	    #INVERT := NOT #INVERT;
	END_IF;
	
	IF #tr.N AND #allowed_change THEN
	    #SR := false;
	    #RS := true;
	    
	    #R := false;
	END_IF;
	
	IF #tr_al.N AND #allowed_change THEN
	    #SR := false;
	    #RS := true;
	    #R := false;
	    #INVERT := false;
	END_IF;
	
	#N := #tr_al.N OR #tr.N;
	
	#changed := #tr.N OR #tr.P;
END_FUNCTION_BLOCK

FUNCTION "swap_a_b_f" : Void
{ S7_Optimized_Access := 'TRUE' }
VERSION : 0.1
   VAR_IN_OUT 
      A : Real;
      B : Real;
   END_VAR

   VAR_TEMP 
      buf : Real;
   END_VAR


BEGIN
	
	#buf := #A;
	#A := #B;
	#B := #buf;
END_FUNCTION

FUNCTION_BLOCK "toggle"
{ S7_Optimized_Access := 'TRUE' }
VERSION : 0.1
   VAR_INPUT 
      flip : Bool;
   END_VAR

   VAR_IN_OUT 
      InOut : Bool;
   END_VAR

   VAR 
      flip_was : Bool;
   END_VAR


BEGIN
	IF #flip AND NOT #flip_was THEN
	    #InOut := NOT #InOut;
	END_IF;
	#flip_was := #flip;
	    
END_FUNCTION_BLOCK

FUNCTION "f_ai" : Real
{ S7_Optimized_Access := 'TRUE' }
VERSION : 0.1
   VAR_INPUT 
      in : Int;
   END_VAR


BEGIN
	#f_ai:=INT_TO_REAL(#in)*10.0 /27632.0;
END_FUNCTION

FUNCTION_BLOCK "INC_limited"
{ S7_Optimized_Access := 'TRUE' }
VERSION : 0.1
   VAR_INPUT 
      CLK : Bool;
      N : Int;
   END_VAR

   VAR_IN_OUT 
      I : Int;
   END_VAR

   VAR 
      mem : Bool;
   END_VAR


BEGIN
	IF #CLK AND NOT #mem THEN
	    #I := (#I + 1)MOD #N;
	END_IF;
	#mem := #CLK;
	    
END_FUNCTION_BLOCK

FUNCTION_BLOCK "TRIGA"
{ S7_Optimized_Access := 'TRUE' }
VERSION : 0.1
   VAR_INPUT 
      CLK : Bool;
   END_VAR

   VAR_OUTPUT 
      P : Bool;
      N : Bool;
   END_VAR

   VAR 
      mem : Bool;
   END_VAR


BEGIN
	#P := #CLK AND NOT #mem;
	#N := NOT #CLK AND #mem;
	
	#mem := #CLK;
END_FUNCTION_BLOCK

DATA_BLOCK "deletemot_speed_wdir_slowly_accelerated_DB"   // DB39
VERSION : 0.1
// stored: AutoNumber true, DBAccessibleFromOPCUA true, InstanceOfName mot_speed_wdir_slowly_accelerated, InstanceOfType FB
"mot_speed_wdir_slowly_accelerated"
BEGIN
END_DATA_BLOCK

DATA_BLOCK "LIVE_BLINK_MONITOR_DB"   // DB57
VERSION : 0.1
// stored: AutoNumber true, DBAccessibleFromOPCUA true, InstanceOfName LIVE_BLINK_MONITOR, InstanceOfType FB
"LIVE_BLINK_MONITOR"
BEGIN
END_DATA_BLOCK

DATA_BLOCK "lightColumn_DB"   // DB48
VERSION : 0.1
// stored: AutoNumber true, DBAccessibleFromOPCUA true, InstanceOfName lightColumn, InstanceOfType FB
"lightColumn"
BEGIN
END_DATA_BLOCK

DATA_BLOCK "monitor_perifery_DB"   // DB15
VERSION : 0.1
// stored: AutoNumber true, DBAccessibleFromOPCUA true, InstanceOfName monitor_perifery, InstanceOfType FB
"monitor_perifery"
BEGIN
END_DATA_BLOCK

DATA_BLOCK "НулевыеБлокировки_DB"   // DB56
VERSION : 0.1
// stored: AutoNumber true, DBAccessibleFromOPCUA true, InstanceOfName НулевыеБлокировки, InstanceOfType FB
"НулевыеБлокировки"
BEGIN
END_DATA_BLOCK

DATA_BLOCK "BLINKER_PC_DB"   // DB55
VERSION : 0.1
// stored: AutoNumber true, DBAccessibleFromOPCUA true, InstanceOfName BLINKER, InstanceOfType FB
"BLINKER"
BEGIN
END_DATA_BLOCK

DATA_BLOCK "ER_0_root"   // DB11
VERSION : 0.1
// stored: AutoNumber true, DBAccessibleFromOPCUA true, InstanceOfName ER_WN__root_FB, InstanceOfType FB
"ER_WN__root_FB"
BEGIN
END_DATA_BLOCK

DATA_BLOCK "ER_HMI_btnColor_DB"   // DB9
VERSION : 0.1
// stored: AutoNumber true, DBAccessibleFromOPCUA true, InstanceOfName ER_HMI_btnColor, InstanceOfType FB
"ER_HMI_btnColor"
BEGIN
END_DATA_BLOCK

DATA_BLOCK "ER_SIREN_ON_WNER_count_change"   // DB41
VERSION : 0.1
// stored: AutoNumber true, DBAccessibleFromOPCUA true, InstanceOfName I_TRIG_int_change, InstanceOfType FB
"I_TRIG_int_change"
BEGIN
END_DATA_BLOCK

DATA_BLOCK "WN_0_root"   // DB7
VERSION : 0.1
// stored: AutoNumber true, DBAccessibleFromOPCUA true, InstanceOfName ER_WN__root_FB, InstanceOfType FB
"ER_WN__root_FB"
BEGIN
END_DATA_BLOCK

DATA_BLOCK "blinker_LEDDESK"   // DB25
VERSION : 0.1
// stored: AutoNumber true, DBAccessibleFromOPCUA true, InstanceOfName BLINKER, InstanceOfType FB
"BLINKER"
BEGIN
END_DATA_BLOCK

DATA_BLOCK "LightBarrier_DB"   // DB74
VERSION : 0.1
// stored: AutoNumber true, DBAccessibleFromOPCUA true, InstanceOfName LightBarrier, InstanceOfType FB
"LightBarrier"
BEGIN
END_DATA_BLOCK

DATA_BLOCK "Xray_related_FB_DB"   // DB16
VERSION : 0.1
// stored: AutoNumber true, DBAccessibleFromOPCUA true, InstanceOfName Xray_related_FB, InstanceOfType FB
"Xray_related_FB"
BEGIN
END_DATA_BLOCK

DATA_BLOCK "laser_centering_device_DB"   // DB4
VERSION : 0.1
// stored: AutoNumber true, DBAccessibleFromOPCUA true, InstanceOfName laser_centering_device, InstanceOfType FB
"laser_centering_device"
BEGIN
END_DATA_BLOCK

DATA_BLOCK "magnet__DB"   // DB70
VERSION : 0.1
// stored: AutoNumber true, DBAccessibleFromOPCUA true, InstanceOfName magnet_, InstanceOfType FB
"magnet_"
BEGIN
END_DATA_BLOCK

DATA_BLOCK "shutter_DB"   // DB47
VERSION : 0.1
// stored: AutoNumber true, DBAccessibleFromOPCUA true, InstanceOfName shutter, InstanceOfType FB
"shutter"
BEGIN
END_DATA_BLOCK

DATA_BLOCK "M1Z"   // DB13
VERSION : 0.1
// stored: AutoNumber true, DBAccessibleFromOPCUA true, InstanceOfName axis_FBD, InstanceOfType FB
"axis_FBD"
BEGIN
END_DATA_BLOCK

DATA_BLOCK "M2Y"   // DB14
VERSION : 0.1
// stored: AutoNumber true, DBAccessibleFromOPCUA true, InstanceOfName axis_FBD, InstanceOfType FB
"axis_FBD"
BEGIN
END_DATA_BLOCK

DATA_BLOCK "M3X"   // DB20
VERSION : 0.1
// stored: AutoNumber true, DBAccessibleFromOPCUA true, InstanceOfName axis_FBD, InstanceOfType FB
"axis_FBD"
BEGIN
END_DATA_BLOCK

DATA_BLOCK "M4O1tilt"   // DB21
VERSION : 0.1
// stored: AutoNumber true, DBAccessibleFromOPCUA true, InstanceOfName axis_FBD, InstanceOfType FB
"axis_FBD"
BEGIN
END_DATA_BLOCK

DATA_BLOCK "M5O2rot"   // DB22
VERSION : 0.1
// stored: AutoNumber true, DBAccessibleFromOPCUA true, InstanceOfName axis_FBD, InstanceOfType FB
"axis_FBD"
BEGIN
END_DATA_BLOCK

DATA_BLOCK "M6doors"   // DB26
VERSION : 0.1
// stored: AutoNumber true, DBAccessibleFromOPCUA true, InstanceOfName axis_FBD, InstanceOfType FB
"axis_FBD"
BEGIN
END_DATA_BLOCK

DATA_BLOCK "_BTNS"   // DB3
VERSION : 0.1
// stored: AutoNumber true, DBAccessibleFromOPCUA true, InstanceOfName BTNS_FB, InstanceOfType FB
"BTNS_FB"
BEGIN
END_DATA_BLOCK

DATA_BLOCK "_DOOORS"   // DB71
VERSION : 0.1
// stored: AutoNumber true, DBAccessibleFromOPCUA true, InstanceOfName _DOOORS_fb, InstanceOfType FB
"_DOOORS_fb"
BEGIN
END_DATA_BLOCK

DATA_BLOCK "artLimFormer_DB"   // DB73
VERSION : 0.1
// stored: AutoNumber true, DBAccessibleFromOPCUA true, InstanceOfName artLimFormer, InstanceOfType FB
"artLimFormer"
BEGIN
END_DATA_BLOCK

DATA_BLOCK "delete"   // DB72
VERSION : 0.1
// stored: AutoNumber true, DBAccessibleFromOPCUA true, InstanceOfName artLimiter, InstanceOfType FB
"artLimiter"
BEGIN
END_DATA_BLOCK

DATA_BLOCK "edelete"   // DB77
VERSION : 0.1
// stored: AutoNumber true, DBAccessibleFromOPCUA true, InstanceOfName Cycle_iterator_spot_generator, InstanceOfType FB
"Cycle_iterator_spot_generator"
BEGIN
END_DATA_BLOCK

DATA_BLOCK "Block_1_DB"   // DB62
VERSION : 0.1
// stored: AutoNumber true, DBAccessibleFromOPCUA true, InstanceOfName _ML2_ts_block1, InstanceOfType FB
"_ML2_ts_block1"
BEGIN
END_DATA_BLOCK

DATA_BLOCK "Cycle_iterator_spot_generator_DB"   // DB78
VERSION : 0.1
// stored: AutoNumber true, DBAccessibleFromOPCUA true, InstanceOfName Cycle_iterator_spot_generator, InstanceOfType FB
"Cycle_iterator_spot_generator"
BEGIN
END_DATA_BLOCK

DATA_BLOCK "DELETEw"   // DB58
VERSION : 0.1
// stored: AutoNumber true, DBAccessibleFromOPCUA true, InstanceOfName _spot_iteratorWaitForXray, InstanceOfType FB
"_spot_iteratorWaitForXray"
BEGIN
END_DATA_BLOCK

DATA_BLOCK "_ML2_modeDB"   // DB12
VERSION : 0.1
// stored: AutoNumber true, DBAccessibleFromOPCUA true, InstanceOfName _ML2_mode, InstanceOfType FB
"_ML2_mode"
BEGIN
END_DATA_BLOCK

DATA_BLOCK "_ML2_target_supplierDB"   // DB30
VERSION : 0.1
// stored: AutoNumber true, DBAccessibleFromOPCUA true, InstanceOfName _ML2_target_supplier, InstanceOfType FB
"_ML2_target_supplier"
BEGIN
   HomePos.M1Z := 110.0;
   HomePos.M2Y := 700.0;
   HomePos.M3X := 670.0;
   HomePos.M4O1 := 50.0;
   HomePos.M5O2 := 300.0;
   LoadPos.M1Z := 110.0;
   LoadPos.M2Y := 700.0;
   LoadPos.M3X := 670.0;
   LoadPos.M4O1 := 50.0;
   LoadPos.M5O2 := 300.0;
END_DATA_BLOCK

DATA_BLOCK "defects_util_DB"   // DB37
VERSION : 0.1
// stored: AutoNumber true, DBAccessibleFromOPCUA true, InstanceOfName defects_util, InstanceOfType FB
"defects_util"
BEGIN
END_DATA_BLOCK

DATA_BLOCK "delete2"   // DB59
VERSION : 0.1
// stored: AutoNumber true, DBAccessibleFromOPCUA true, InstanceOfName _ML2_target_supplier, InstanceOfType FB
"_ML2_target_supplier"
BEGIN
   Spots_pos_AR.N := 4;
   Spots_pos_AR.pos_AR[1].M1Z := 11.0;
   Spots_pos_AR.pos_AR[2].M1Z := 33.0;
   Spots_pos_AR.pos_AR[3].M1Z := 55.0;
   Spots_pos_AR.pos_AR[4].M1Z := 44.0;
   Spots_pos_AR.pos_AR[5..30].M1Z := 0.0;
   Spots_pos_AR.pos_AR[1..30].M2Y := 0.0;
   Spots_pos_AR.pos_AR[1..30].M3X := 0.0;
   Spots_pos_AR.pos_AR[1..30].M4O1 := 0.0;
   Spots_pos_AR.pos_AR[1..30].M5O2 := 0.0;
   CurPositios.M1Z := 0.0;
   CurPositios.M2Y := 0.0;
   CurPositios.M3X := 0.0;
   CurPositios.M4O1 := 0.0;
   CurPositios.M5O2 := 0.0;
   def_util_db.xBdefect_inc := FALSE;
   def_util_db.xBdefect_dec := FALSE;
   def_util_db.xDefectsClearAll := FALSE;
   def_util_db.xDefect_Save := FALSE;
   def_util_db.positions.M1Z := 0.0;
   def_util_db.positions.M2Y := 0.0;
   def_util_db.positions.M3X := 0.0;
   def_util_db.positions.M4O1 := 0.0;
   def_util_db.positions.M5O2 := 0.0;
   def_util_db.go_to_defect_now := FALSE;
   def_util_db.xyBeepDone := FALSE;
   def_util_db.mem1 := FALSE;
   def_util_db.mem2 := FALSE;
   def_util_db.xdefect_dec_was := FALSE;
   def_util_db.xdefect_inc_was := FALSE;
   def_util_db.xDefect_Save_was := FALSE;
   def_util_db.xDefectsClearAll_was := FALSE;
END_DATA_BLOCK

DATA_BLOCK "delete_ML2_target_supplier_DB"   // DB63
VERSION : 0.1
// stored: AutoNumber true, DBAccessibleFromOPCUA true, InstanceOfName _ML2_target_supplier, InstanceOfType FB
"_ML2_target_supplier"
BEGIN
END_DATA_BLOCK

DATA_BLOCK "deleteeeaman_sel_target_DB"   // DB52
VERSION : 0.1
// stored: AutoNumber true, DBAccessibleFromOPCUA true, InstanceOfName aman_sel_target, InstanceOfType FB
"aman_sel_target"
BEGIN
END_DATA_BLOCK

DATA_BLOCK "deleter"   // DB66
VERSION : 0.1
// stored: AutoNumber true, DBAccessibleFromOPCUA true, InstanceOfName _ML2_ts_block1, InstanceOfType FB
"_ML2_ts_block1"
BEGIN
END_DATA_BLOCK

DATA_BLOCK "execute_semiauto_DB"   // DB36
VERSION : 0.1
// stored: AutoNumber true, DBAccessibleFromOPCUA true, InstanceOfName execute_semiauto, InstanceOfType FB
"execute_semiauto"
BEGIN
END_DATA_BLOCK

DATA_BLOCK "not_used_blocks_DB"   // DB68
VERSION : 0.1
// stored: AutoNumber true, DBAccessibleFromOPCUA true, InstanceOfName not_used_blocks, InstanceOfType FB
"not_used_blocks"
BEGIN
END_DATA_BLOCK

DATA_BLOCK "HomePosManagerDb"   // DB65
VERSION : 0.1
// stored: AutoNumber true, DBAccessibleFromOPCUA true, InstanceOfName _hmi_singleSpotManager, InstanceOfType FB
"_hmi_singleSpotManager"
BEGIN
END_DATA_BLOCK

DATA_BLOCK "Load_pos_managerDB"   // DB64
VERSION : 0.1
// stored: AutoNumber true, DBAccessibleFromOPCUA true, InstanceOfName _hmi_singleSpotManager, InstanceOfType FB
"_hmi_singleSpotManager"
BEGIN
END_DATA_BLOCK

DATA_BLOCK "_hmi_spot_manager_DB"   // DB51
VERSION : 0.1
// stored: AutoNumber true, DBAccessibleFromOPCUA true, InstanceOfName _hmi_spot_manager, InstanceOfType FB
"_hmi_spot_manager"
BEGIN
END_DATA_BLOCK

DATA_BLOCK "control1PosManagerDB"   // DB79
VERSION : 0.1
// stored: AutoNumber true, DBAccessibleFromOPCUA true, InstanceOfName _hmi_singleSpotManager, InstanceOfType FB
"_hmi_singleSpotManager"
BEGIN
END_DATA_BLOCK

DATA_BLOCK "control2PosManagerDB"   // DB80
VERSION : 0.1
// stored: AutoNumber true, DBAccessibleFromOPCUA true, InstanceOfName _hmi_singleSpotManager, InstanceOfType FB
"_hmi_singleSpotManager"
BEGIN
END_DATA_BLOCK

DATA_BLOCK "_screen_home_DB"   // DB75
VERSION : 0.1
// stored: AutoNumber true, DBAccessibleFromOPCUA true, InstanceOfName _screen_Targets, InstanceOfType FB
"_screen_Targets"
BEGIN
END_DATA_BLOCK

DATA_BLOCK "ER_0ESTOPS"   // DB43
VERSION : 0.1
// stored: AutoNumber true, DBAccessibleFromOPCUA true, InstanceOfName ER_WORD, InstanceOfType FB
"ER_WORD"
BEGIN
END_DATA_BLOCK

DATA_BLOCK "ER_1AxisMain"   // DB35
VERSION : 0.1
// stored: AutoNumber true, DBAccessibleFromOPCUA true, InstanceOfName ER_WORD, InstanceOfType FB
"ER_WORD"
BEGIN
END_DATA_BLOCK

DATA_BLOCK "ER_1DESK"   // DB50
VERSION : 0.1
// stored: AutoNumber true, DBAccessibleFromOPCUA true, InstanceOfName ER_WORD, InstanceOfType FB
"ER_WORD"
BEGIN
END_DATA_BLOCK

DATA_BLOCK "WN_0ESTOPS"   // DB24
VERSION : 0.1
// stored: AutoNumber true, DBAccessibleFromOPCUA true, InstanceOfName ER_WORD, InstanceOfType FB
"ER_WORD"
BEGIN
END_DATA_BLOCK

DATA_BLOCK "WN_1Xray"   // DB49
VERSION : 0.1
// stored: AutoNumber true, DBAccessibleFromOPCUA true, InstanceOfName ER_WORD, InstanceOfType FB
"ER_WORD"
BEGIN
END_DATA_BLOCK

DATA_BLOCK "WN_2AxisMain"   // DB34
VERSION : 0.1
// stored: AutoNumber true, DBAccessibleFromOPCUA true, InstanceOfName ER_WORD, InstanceOfType FB
"ER_WORD"
BEGIN
END_DATA_BLOCK

DATA_BLOCK "WN_4PC"   // DB54
VERSION : 0.1
// stored: AutoNumber true, DBAccessibleFromOPCUA true, InstanceOfName ER_WORD, InstanceOfType FB
"ER_WORD"
BEGIN
END_DATA_BLOCK

DATA_BLOCK "wn_5auto"   // DB38
VERSION : 0.1
// stored: AutoNumber true, DBAccessibleFromOPCUA true, InstanceOfName ER_WORD, InstanceOfType FB
"ER_WORD"
BEGIN
END_DATA_BLOCK

DATA_BLOCK "er_ack_ton"   // DB31
{ S7_Optimized_Access := 'TRUE' }
// stored: AutoNumber true, DBAccessibleFromOPCUA true, InstanceOfName IEC_TIMER, OfSystemLibElement IEC_TIMER, OfSystemLibVersion 1.0
"IEC_TIMER"
   // VAR
   //    PT : Time;
   //    ET { ExternalWritable := 'False'} : Time;
   //    IN : Bool;
   //    Q { ExternalWritable := 'False'} : Bool;
   // END_VAR
BEGIN
END_DATA_BLOCK

DATA_BLOCK "tonBuz_alarm"   // DB42
{ S7_Optimized_Access := 'TRUE' }
// stored: AutoNumber true, DBAccessibleFromOPCUA true, InstanceOfName IEC_TIMER, OfSystemLibElement IEC_TIMER, OfSystemLibVersion 1.0
"IEC_TIMER"
   // VAR
   //    PT : Time;
   //    ET { ExternalWritable := 'False'} : Time;
   //    IN : Bool;
   //    Q { ExternalWritable := 'False'} : Bool;
   // END_VAR
BEGIN
END_DATA_BLOCK

DATA_BLOCK "CAB_yLEDALARM_DB"   // DB45
VERSION : 0.1
// stored: AutoNumber true, DBAccessibleFromOPCUA true, InstanceOfName LED_FBD, InstanceOfType FB
"LED_FBD"
BEGIN
END_DATA_BLOCK

DATA_BLOCK "LED_lampTestAtStartup_DB"   // DB8
VERSION : 0.1
// stored: AutoNumber true, DBAccessibleFromOPCUA true, InstanceOfName LED_lampTestAtStartup, InstanceOfType FB
"LED_lampTestAtStartup"
BEGIN
END_DATA_BLOCK

DATA_BLOCK "desk_yBUZDoneDB"   // DB6
VERSION : 0.1
// stored: AutoNumber true, DBAccessibleFromOPCUA true, InstanceOfName LED_FBD, InstanceOfType FB
"LED_FBD"
BEGIN
END_DATA_BLOCK

DATA_BLOCK "desk_yBuzAlarmDB"   // DB5
VERSION : 0.1
// stored: AutoNumber true, DBAccessibleFromOPCUA true, InstanceOfName LED_FBD, InstanceOfType FB
"LED_FBD"
BEGIN
END_DATA_BLOCK

DATA_BLOCK "desk_yledAutoDB"   // DB2
VERSION : 0.1
// stored: AutoNumber true, DBAccessibleFromOPCUA true, InstanceOfName LED_FBD, InstanceOfType FB
"LED_FBD"
BEGIN
END_DATA_BLOCK

DATA_BLOCK "MOT1_remSel"   // DB18
VERSION : 0.1
// stored: AutoNumber true, DBAccessibleFromOPCUA true, InstanceOfName axis_manager, InstanceOfType FB
"axis_manager"
BEGIN
END_DATA_BLOCK

DATA_BLOCK "MOT2_remSel"   // DB19
VERSION : 0.1
// stored: AutoNumber true, DBAccessibleFromOPCUA true, InstanceOfName axis_manager, InstanceOfType FB
"axis_manager"
BEGIN
END_DATA_BLOCK

DATA_BLOCK "_spot_iterator"   // DB27
VERSION : 0.1
// stored: AutoNumber true, DBAccessibleFromOPCUA true, InstanceOfName _spot_iteratorWaitForXray, InstanceOfType FB
"_spot_iteratorWaitForXray"
BEGIN
END_DATA_BLOCK

DATA_BLOCK "MAN_DESCRETE_cycle_DB"   // DB32
VERSION : 0.1
// stored: AutoNumber true, DBAccessibleFromOPCUA true, InstanceOfName MAN_DESCRETE_cycle, InstanceOfType FB
"MAN_DESCRETE_cycle"
BEGIN
END_DATA_BLOCK

DATA_BLOCK "man_descrete_sr_DB"   // DB28
VERSION : 0.1
// stored: AutoNumber true, DBAccessibleFromOPCUA true, InstanceOfName man_descrete_sr, InstanceOfType FB
"man_descrete_sr"
BEGIN
END_DATA_BLOCK

DATA_BLOCK "man_desk_button_cell_DB"   // DB29
VERSION : 0.1
// stored: AutoNumber true, DBAccessibleFromOPCUA true, InstanceOfName _ML2_target_supplier, InstanceOfType FB
"_ML2_target_supplier"
BEGIN
END_DATA_BLOCK
